// TIA Portal V19 export
FUNCTION "Pb_Drain_Tank" : Void   // FC64, STL
TITLE = Pb - START/STOP DRAIN TANK
{ S7_Optimized_Access := 'TRUE' }
NAME : PBDRAIN
VERSION : 0.0
// Comment
// stored: AutoNumber false
   VAR_TEMP
      alarmbit : Int;
   END_VAR
BEGIN

NETWORK
TITLE = Pb - START/STOP DRAIN TANK
      AN    "LEDAssignment".K6_BUTTON;  //"PbK6DrainTank"
      BEC;
      R     "LEDAssignment".K6_BUTTON;  // "PbK6DrainTank"
      A     "DUMMY UPD.DRAIN TANK";
      JC    M001;
      O     "S0 PRESTERILIZING";
      O     "S0 CIP TANK";
      S     "ProcessAndPbAlarms"."A"[13];  //A13_DrainTankNotAllowed// drain tank not allowed
      L     13;
      JC    Alrm;

//      BEC
      S     "MY0111";
      S     "MY0112";
      S     "MY0113";
      S     "MY0114";
      S     "LEDAssignment".K6_FLASH;  //"FLASH_K6_DRAIN_TANK"
      S     "LEDAssignment".K6_LIGHT;  //"LIGHT_K6_DRAIN_TANK"
      L     "Setpoints".PT0167SpProduction;  // "DB SETPOINTS".PT0167SpProduction
      T     "STP_PT0167/IP0149_50".PT0167SpSTP;
      S     "AutoPT0167/IP0149";
      S     "DUMMY UPD.DRAIN TANK";
      BEU;
M001: R     "DUMMY UPD.DRAIN TANK";
      R     "MY0112";
      R     "MY0113";
      R     "LEDAssignment".K6_FLASH;  // "FLASH_K6_DRAIN_TANK"
      R     "LEDAssignment".K6_LIGHT;  //"LIGHT_K6_DRAIN_TANK"
      A     "TANK AUTO";
      BEC;
      R     "MY0111";  // IF A-TANK IN PRODUCTION DON'T CLOSE VALVE 01.11
      R     "AutoPT0167/IP0149";
      R     "MY0114";
      BEU;

NETWORK
TITLE = Blockings alarm text
// Blockings alarm
Alrm: NOP   1;
      T     #alarmbit;
      CALL  "Set_Pop_Up_Blocking"
      ( alarmTextNum := #alarmbit
      );  // start blockings text


END_FUNCTION
